FUNCTION_BLOCK FB_ReadAmsValue
VAR_INPUT
	tUpdate					:	TIME 				:=T#900MS;
	
	sNetId					:	T_AmsNetId			:='';
	nPort					:	T_AmsPort			:=851;
	sVarName				:	STRING(255)			:='';
	nDestAddr				:	PVOID;
	nDestLen				:	UDINT;
	tReadTimeout			:	TIME				:=T#2000MS;
	
END_VAR

VAR_OUTPUT
	bReadError		: BOOL := FALSE;
	nReadErrorId	: UDINT;
	
END_VAR

VAR
	
	ET_Read			: TIME := T#0MS;
	bReadEnable		: BOOL := FALSE;
	readBusy		: BOOL := FALSE;
	
	TON_Read		: TON;
	fb_reader	: FB_ReadAdsSymByName;
END_VAR

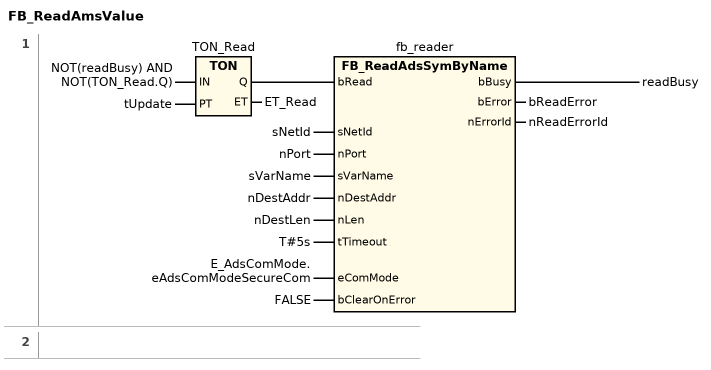
// NETWORK 1
TON_Read(IN := NOT(readBusy) AND NOT(TON_Read.Q), PT := tUpdate, ET => ET_Read); // TON
fb_reader(
    bRead := TON_Read.Q,
    sNetId := sNetId,
    nPort := nPort,
    sVarName := sVarName,
    nDestAddr := nDestAddr,
    nLen := nDestLen,
    tTimeout := T#5s,
    eComMode := E_AdsComMode.eAdsComModeSecureCom,
    bClearOnError := FALSE,
    bError => bReadError,
    nErrorId => nReadErrorId); // FB_ReadAdsSymByName
readBusy := fb_reader.bBusy;

// NETWORK 2

END_FUNCTION_BLOCK

(* stored: Version 1.1.0.1, ProductVersion 3.1.4024.11
   POU FB_ReadAmsValue: Id {3059acc9-03f7-42e5-b9bb-86ef7606208b}, SpecialFunc None *)
